Universal Robots PolyScope program: 27- force_simple.urp

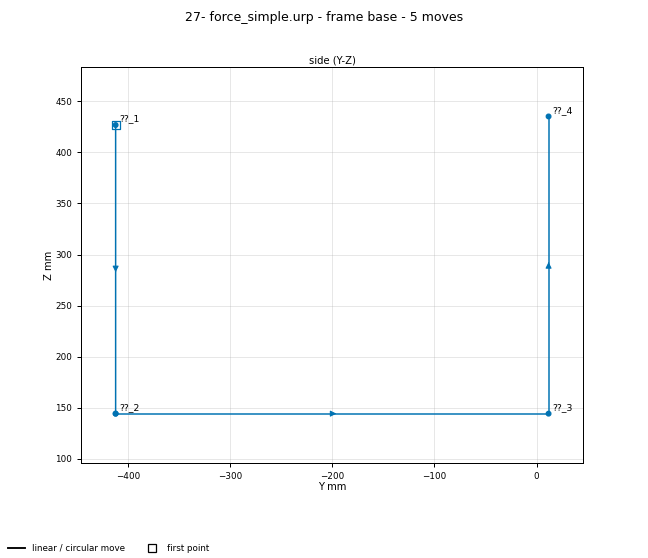
[picture p0: tool path of 27- force_simple.urp in frame base, 5 of 5 moves have a stored position in this frame; points joined in program order, loops and branches not executed]
ProgramRoot directory=/home/ur/ursim-3.1/programs/basic training/27- force_simple; kinematics=(a=[0, -0.425, -0.39225, 0, 0, 0], d=[0.08916, 0, 0, 0.10915, 0.09465, 0.0823], alpha=[1.5708, 0, 0, 1.5708, -1.5708, 0], deltaTheta=[0, 0, 0, 0, 0, 0], status=notInitialized); lastSavedInVersion=(project__name=Polyscope, major__version=3, minor__version=1, svn__revision=17195, build__date=Mar 11 2015, 13:02:28); name=27- force_simple; programVersion=(project__name=Polyscope, major__version=3, minor__version=1, svn__revision=17195, build__date=Mar 11 2015, 13:02:28); robotEnvironmentFileName=default; serialNumberRobot=2014350001
  MainProgram cartesianAcceleration=1.2; cartesianSpeed=0.25; jointAcceleration=1.3962634015954636; jointSpeed=1.0471975511965976; sharedProcessMoveBlendRadius=0.025; motionType=JOINT_SPACE
    Move cartesianAcceleration=1.2; cartesianSpeed=0.25; jointAcceleration=1.3962634015954636; jointSpeed=1.0471975511965976; sharedProcessMoveBlendRadius=0.025; motionType=CARTESIAN_SPACE
      Waypoint blendRadius=0.05; cartesianAcceleration=1.2; cartesianSpeed=0.25; jointAcceleration=1.3962634015954636; jointSpeed=1.0471975511965976; nextMotionTime=2.0; stoppoint=true; useSharedBlendParameter=true; useSharedParameters=true; outputFlangePose=(pos=(x=0.31381586839482134, y=-0.4119515970671896, z=0.4267139361837215), rot=(x=-0.0012211004006276967, y=3.116276455539744, z=0.03889228887857356)); position=TCP in base x=313.816 y=-411.952 z=426.714 mm, rx=-0.0012 ry=3.1163 rz=0.0389 rad; joints [-40.862, -92.666, -88.063, -89.122, 92.021, 49.096] deg; positionType=FIXED_POSITION; waypointPoseInFeatureCoordinates=(pos=(x=0.31381590983180896, y=-0.4119516485752222, z=0.42671398574289104), rot=(x=-0.0012210227574820896, y=3.1162763421843955, z=0.03889217574521001)); name=路点_1
      Waypoint blendRadius=0.05; cartesianAcceleration=1.2; cartesianSpeed=0.25; jointAcceleration=1.3962634015954636; jointSpeed=1.0471975511965976; nextMotionTime=2.0; stoppoint=true; useSharedBlendParameter=true; useSharedParameters=true; outputFlangePose=(pos=(x=0.31381579772272766, y=-0.4119515359318888, z=0.1442953136694916), rot=(x=-0.0012211004005269902, y=3.116276455539779, z=0.03889228887864879)); position=TCP in base x=313.816 y=-411.952 z=144.295 mm, rx=-0.0012 ry=3.1163 rz=0.0389 rad; joints [-40.862, -107.276, -115.96, -46.614, 92.021, 49.096] deg; positionType=FIXED_POSITION; waypointPoseInFeatureCoordinates=(pos=(x=0.31381578975528135, y=-0.41195154462597217, z=0.1442953615523033), rot=(x=-0.0012210227574823039, y=3.1162763421843898, z=0.0388921757452197)); name=路点_2
      Force force__mode__wrench=[0, 0, 20, 0, 0, 0]; limits__force=[0.15, 0.15, 0.15, 1.0472, 1.0472, 1.0472]; limits__motion=[0.1, 0.1, 0.1, 0.34907, 0.34907, 0.34907]; selection__vector=[0, 0, 1, 0, 0, 0]; type=FORCE_TYPE_SIMPLE
        Waypoint blendRadius=0.05; cartesianAcceleration=1.2; cartesianSpeed=0.25; jointAcceleration=1.3962634015954636; jointSpeed=1.0471975511965976; nextMotionTime=2.0; stoppoint=true; useSharedBlendParameter=true; useSharedParameters=true; outputFlangePose=(pos=(x=0.31381579772272766, y=-0.4119515359318888, z=0.1442953136694916), rot=(x=-0.0012211004005269902, y=3.116276455539779, z=0.03889228887864879)); position=TCP in base x=313.816 y=-411.952 z=144.295 mm, rx=-0.0012 ry=3.1163 rz=0.0389 rad; joints [-40.862, -107.276, -115.96, -46.614, 92.021, 49.096] deg; positionType=FIXED_POSITION; waypointPoseInFeatureCoordinates=(pos=(x=0.31381578975528135, y=-0.41195154462597217, z=0.1442953615523033), rot=(x=-0.0012210227574823039, y=3.1162763421843898, z=0.0388921757452197)); name=路点_2
        Waypoint blendRadius=0.05; cartesianAcceleration=1.2; cartesianSpeed=0.25; jointAcceleration=1.3962634015954636; jointSpeed=1.0471975511965976; nextMotionTime=2.0; stoppoint=true; useSharedBlendParameter=true; useSharedParameters=true; outputFlangePose=(pos=(x=0.3138155851973246, y=0.011667259731930639, z=0.14429536384706224), rot=(x=-0.001221099782200677, y=3.1162764219019112, z=0.03889229581880099)); position=TCP in base x=313.816 y=11.667 z=144.295 mm, rx=-0.0012 ry=3.1163 rz=0.0389 rad; joints [22.25, -80.181, -146.309, -41.639, 90.78, 112.218] deg; positionType=FIXED_POSITION; waypointPoseInFeatureCoordinates=(pos=(x=0.3138155476953759, y=0.01166723946943694, z=0.14429537190157213), rot=(x=-0.0012211116482669958, y=3.116276436312879, z=0.03889222183175042)); name=路点_3
      Waypoint blendRadius=0.05; cartesianAcceleration=1.2; cartesianSpeed=0.25; jointAcceleration=1.3962634015954636; jointSpeed=1.0471975511965976; nextMotionTime=2.0; stoppoint=true; useSharedBlendParameter=true; useSharedParameters=true; outputFlangePose=(pos=(x=0.313815697512705, y=0.011667305682312447, z=0.43511396098586885), rot=(x=-0.0012210997820840286, y=3.116276421901974, z=0.038892295819099434)); position=TCP in base x=313.816 y=11.667 z=435.114 mm, rx=-0.0012 ry=3.1163 rz=0.0389 rad; joints [22.25, -63.147, -110.127, -94.855, 90.78, 112.218] deg; positionType=FIXED_POSITION; waypointPoseInFeatureCoordinates=(pos=(x=0.31381572304967886, y=0.011667311145819413, z=0.43511389864409916), rot=(x=-0.0012211092056726846, y=3.1162766587347694, z=0.03889208400031899)); name=路点_4
